(* PLC project Generated.project, CODESYS CODESYS V3.5 SP19 Patch 1 *)
(* stored: creationDateTime 2026-08-11T18:19:14.764528, modificationDateTime 2026-08-11T18:19:14.764528 *)

(* values of E_CycleStep: INIT: Vérifs cohérence états + sécurités, mise en position init; WORK_POS_SELECT: Choix opérateur pos travail 1/2 + déplacement validé joystick; DESCENDING_OPEN: Plongée benne déjà ouvert, M1+M2 synchro; BOTTOM_TOUCH_WAIT: Attente info BOOL capteur "fond touché"; SYNCHRO_ADJUST: Désynchro M2 petite vitesse (offset X) → fermeture benne; CTRL_ASCENDING: Remontée lente de contrôle (vérification fermeture); ASCENDING_LOADED: Remontée pleine vitesse charge; DRAINING_PAUSE: Égouttage temporisé (durée RETAIN); TRANSLATION_MOVE: Déplacement translation M3 vers trémie; DESCENDING_OPEN_DUMP: Descente de vidage + ouverture benne; RETURN_WORK_POS: Retour position travail (remontée synchro); READY: Cycle terminé, prêt à reboucler; ERROR_HOLD: Arrêt sûr figé sur défaut (SafeStop) *)

{attribute 'qualified_only'}
{attribute 'strict'}
TYPE E_CycleStep : (INIT := 0, WORK_POS_SELECT := 1, DESCENDING_OPEN := 2, BOTTOM_TOUCH_WAIT := 3, SYNCHRO_ADJUST := 4, CTRL_ASCENDING := 5, ASCENDING_LOADED := 6, DRAINING_PAUSE := 7, TRANSLATION_MOVE := 8, DESCENDING_OPEN_DUMP := 9, RETURN_WORK_POS := 10, READY := 11, ERROR_HOLD := 12);
END_TYPE
